// TIA Portal V15.1 export
// export: Created 2024-05-17T05:38:23.9003933Z, ExportSetting WithDefaults, DisplayName Totally Integrated Automation Portal, DisplayVersion V15.1 Update 5, DisplayName TIA Portal Openness, DisplayVersion V15.1 Update 5, DisplayName SINAMICS Startdrive Advanced, DisplayVersion V15.1, DisplayName G130, G150, S120, S150, SINAMICS MV, S210, DisplayVersion V15.1, DisplayName G110M, G120, G120C, G120D, G120P, DisplayVersion V15.1, DisplayName STEP 7 Professional, DisplayVersion V15.1 Update 5, DisplayName STEP 7 Safety, DisplayVersion V15.1, DisplayName WinCC Professional, DisplayVersion V15.1 Update 5, DisplayName SIMATIC Visualization Architect, DisplayVersion V15.1
FUNCTION "F209220ZS01Logic" : Void   // FC7021, F_FBD
TITLE = Safety Inputs ZMProc / Safety Logic 209220ZS01
{ S7_Optimized_Access := 'TRUE' }
VERSION : 0.1
// stored: AutoNumber false, IsIECCheckEnabled false, UDAEnableTagReadback false
   VAR_TEMP   // added for the SCL form of the ladder/FBD networks
      _w1 : Bool;
   END_VAR
BEGIN

REGION Network 1: **** 4.4 - Machine Status - Calculation **** Emergency Stop OK
   // Emergency Stop Ok When All Safety Inputs Are Ok
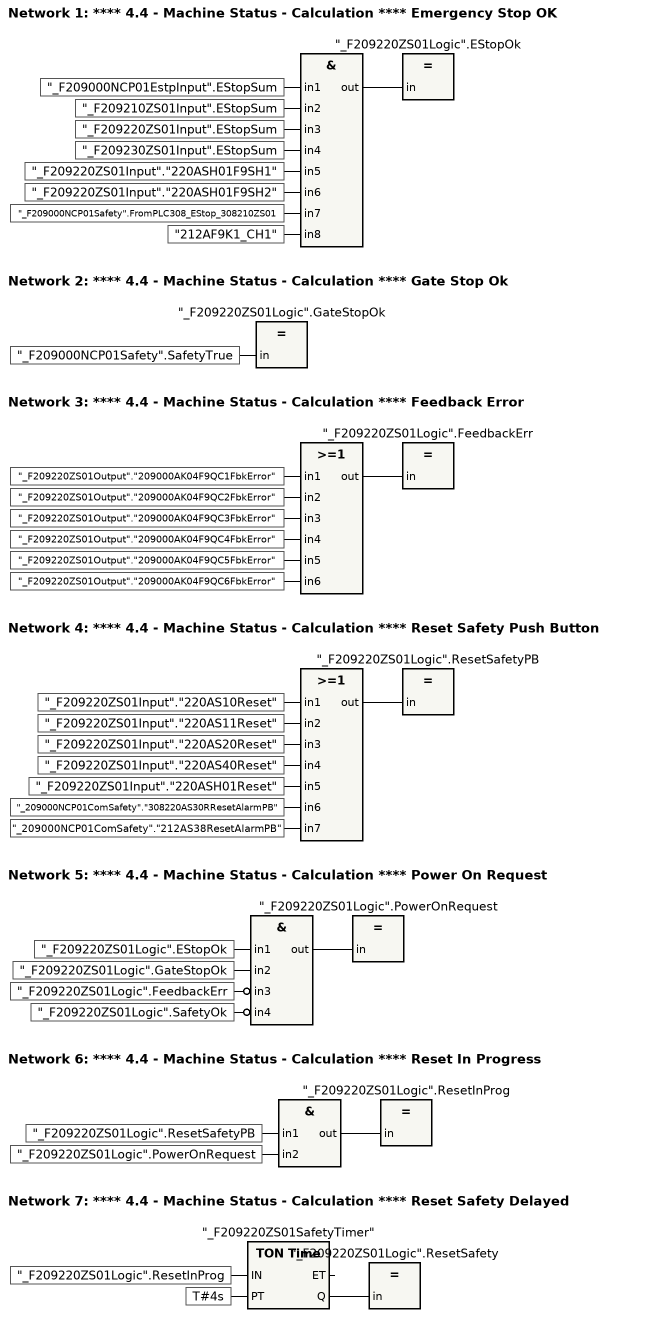
   "_F209220ZS01Logic".EStopOk := "_F209000NCP01EstpInput".EStopSum AND "_F209210ZS01Input".EStopSum AND "_F209220ZS01Input".EStopSum AND "_F209230ZS01Input".EStopSum AND "_F209220ZS01Input"."220ASH01F9SH1" AND "_F209220ZS01Input"."220ASH01F9SH2" AND "_F209000NCP01Safety".FromPLC308_EStop_308210ZS01 AND "212AF9K1_CH1";
END_REGION

REGION Network 2: **** 4.4 - Machine Status - Calculation **** Gate Stop Ok
   // Gate Stop Ok
   "_F209220ZS01Logic".GateStopOk := "_F209000NCP01Safety".SafetyTrue;
END_REGION

REGION Network 3: **** 4.4 - Machine Status - Calculation **** Feedback Error
   // Feedback Error
   "_F209220ZS01Logic".FeedbackErr := "_F209220ZS01Output"."209000AK04F9QC1FbkError" OR "_F209220ZS01Output"."209000AK04F9QC2FbkError" OR "_F209220ZS01Output"."209000AK04F9QC3FbkError" OR "_F209220ZS01Output"."209000AK04F9QC4FbkError" OR "_F209220ZS01Output"."209000AK04F9QC5FbkError" OR "_F209220ZS01Output"."209000AK04F9QC6FbkError";
END_REGION

REGION Network 4: **** 4.4 - Machine Status - Calculation **** Reset Safety Push Button
   // Reset Safety Push Button
   "_F209220ZS01Logic".ResetSafetyPB := "_F209220ZS01Input"."220AS10Reset" OR "_F209220ZS01Input"."220AS11Reset" OR "_F209220ZS01Input"."220AS20Reset" OR "_F209220ZS01Input"."220AS40Reset" OR "_F209220ZS01Input"."220ASH01Reset" OR "_209000NCP01ComSafety"."308220AS30RResetAlarmPB" OR "_209000NCP01ComSafety"."212AS38ResetAlarmPB";
END_REGION

REGION Network 5: **** 4.4 - Machine Status - Calculation **** Power On Request
   // Power On Request
   "_F209220ZS01Logic".PowerOnRequest := "_F209220ZS01Logic".EStopOk AND "_F209220ZS01Logic".GateStopOk AND NOT "_F209220ZS01Logic".FeedbackErr AND NOT "_F209220ZS01Logic".SafetyOk;
END_REGION

REGION Network 6: **** 4.4 - Machine Status - Calculation **** Reset In Progress
   // Reset In Progress
   "_F209220ZS01Logic".ResetInProg := "_F209220ZS01Logic".ResetSafetyPB AND "_F209220ZS01Logic".PowerOnRequest;
END_REGION

REGION Network 7: **** 4.4 - Machine Status - Calculation **** Reset Safety Delayed
   // Reset Safety Delayed
   "_F209220ZS01SafetyTimer".TON(IN := "_F209220ZS01Logic".ResetInProg, PT := T#4s);
   "_F209220ZS01Logic".ResetSafety := "_F209220ZS01SafetyTimer".Q;
END_REGION

REGION Network 8: **** 4.4 - Machine Status - Calculation **** Power On
   // Power On
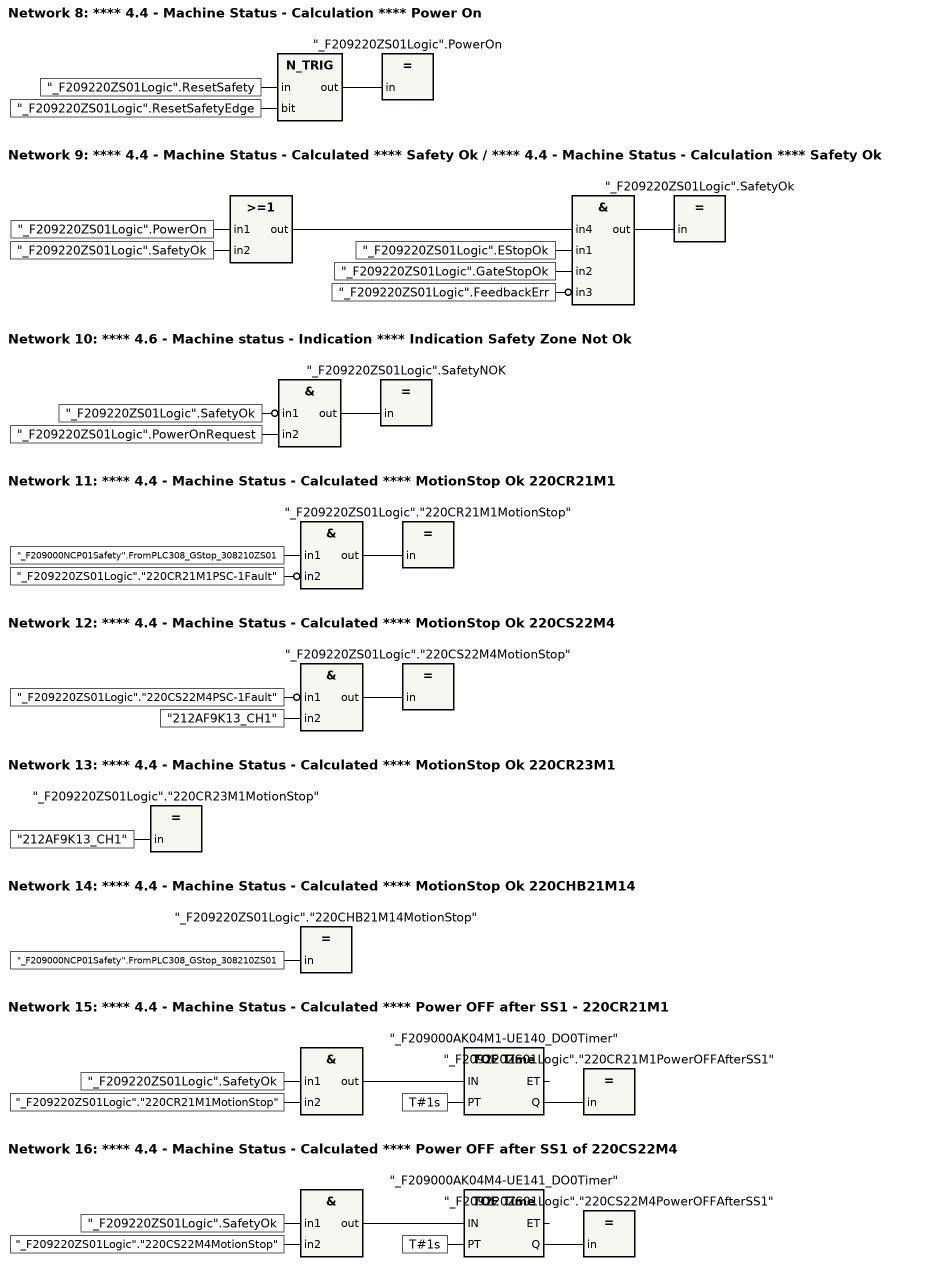
   #_w1 := NOT "_F209220ZS01Logic".ResetSafety AND "_F209220ZS01Logic".ResetSafetyEdge;   // falling edge
   "_F209220ZS01Logic".ResetSafetyEdge := "_F209220ZS01Logic".ResetSafety;
   "_F209220ZS01Logic".PowerOn := #_w1;
END_REGION

REGION Network 9: **** 4.4 - Machine Status - Calculated **** Safety Ok / **** 4.4 - Machine Status - Calculation **** Safety Ok
   // All safety is ok
   "_F209220ZS01Logic".SafetyOk := ("_F209220ZS01Logic".PowerOn OR "_F209220ZS01Logic".SafetyOk) AND "_F209220ZS01Logic".EStopOk AND "_F209220ZS01Logic".GateStopOk AND NOT "_F209220ZS01Logic".FeedbackErr;
END_REGION

REGION Network 10: **** 4.6 - Machine status - Indication **** Indication Safety Zone Not Ok
   // Indication Safety Zone Not Ok
   "_F209220ZS01Logic".SafetyNOK := NOT "_F209220ZS01Logic".SafetyOk AND "_F209220ZS01Logic".PowerOnRequest;
END_REGION

REGION Network 11: **** 4.4 - Machine Status - Calculated **** MotionStop Ok 220CR21M1
   // MotionStop Ok
   "_F209220ZS01Logic"."220CR21M1MotionStop" := "_F209000NCP01Safety".FromPLC308_GStop_308210ZS01 AND NOT "_F209220ZS01Logic"."220CR21M1PSC-1Fault";
END_REGION

REGION Network 12: **** 4.4 - Machine Status - Calculated **** MotionStop Ok 220CS22M4
   // MotionStop Ok
   "_F209220ZS01Logic"."220CS22M4MotionStop" := NOT "_F209220ZS01Logic"."220CS22M4PSC-1Fault" AND "212AF9K13_CH1";
END_REGION

REGION Network 13: **** 4.4 - Machine Status - Calculated **** MotionStop Ok 220CR23M1
   // MotionStop Ok
   "_F209220ZS01Logic"."220CR23M1MotionStop" := "212AF9K13_CH1";
END_REGION

REGION Network 14: **** 4.4 - Machine Status - Calculated **** MotionStop Ok 220CHB21M14
   // MotionStop Ok
   "_F209220ZS01Logic"."220CHB21M14MotionStop" := "_F209000NCP01Safety".FromPLC308_GStop_308210ZS01;
END_REGION

REGION Network 15: **** 4.4 - Machine Status - Calculated **** Power OFF after SS1 - 220CR21M1
   // SEW Drive Delay Power OFF
   "_F209000AK04M1-UE140_DO0Timer".TOF(IN := "_F209220ZS01Logic".SafetyOk AND "_F209220ZS01Logic"."220CR21M1MotionStop",
                           PT := T#1s);
   "_F209220ZS01Logic"."220CR21M1PowerOFFAfterSS1" := "_F209000AK04M1-UE140_DO0Timer".Q;
END_REGION

REGION Network 16: **** 4.4 - Machine Status - Calculated **** Power OFF after SS1 of 220CS22M4
   // SEW Drive Delay Power OFF
   "_F209000AK04M4-UE141_DO0Timer".TOF(IN := "_F209220ZS01Logic".SafetyOk AND "_F209220ZS01Logic"."220CS22M4MotionStop",
                           PT := T#1s);
   "_F209220ZS01Logic"."220CS22M4PowerOFFAfterSS1" := "_F209000AK04M4-UE141_DO0Timer".Q;
END_REGION

REGION Network 17: **** 4.4 - Machine Status - Calculated **** Power OFF after SS1 - 220CR23M1
   // SEW Drive Delay Power OFF
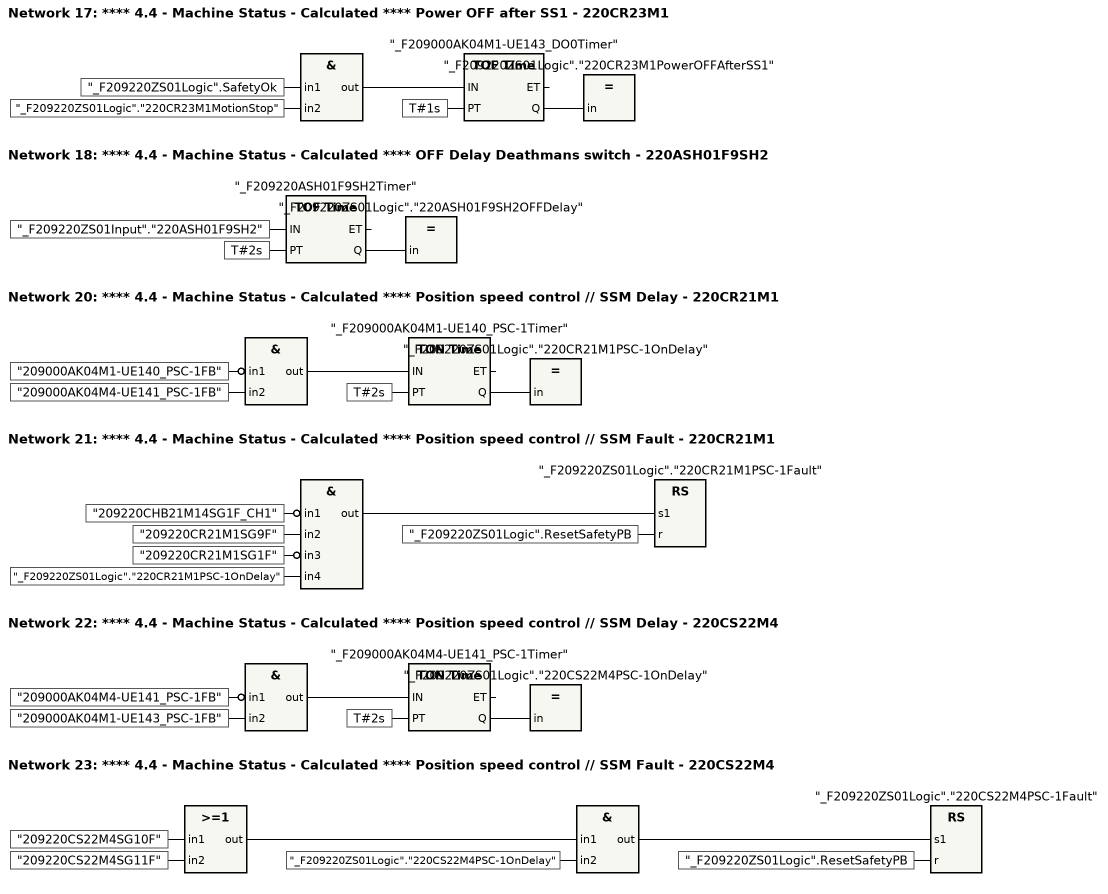
   "_F209000AK04M1-UE143_DO0Timer".TOF(IN := "_F209220ZS01Logic".SafetyOk AND "_F209220ZS01Logic"."220CR23M1MotionStop",
                           PT := T#1s);
   "_F209220ZS01Logic"."220CR23M1PowerOFFAfterSS1" := "_F209000AK04M1-UE143_DO0Timer".Q;
END_REGION

REGION Network 18: **** 4.4 - Machine Status - Calculated **** OFF Delay Deathmans switch - 220ASH01F9SH2
   "_F209220ASH01F9SH2Timer".TOF(IN := "_F209220ZS01Input"."220ASH01F9SH2", PT := T#2s);
   "_F209220ZS01Logic"."220ASH01F9SH2OFFDelay" := "_F209220ASH01F9SH2Timer".Q;
END_REGION

REGION Network 19: **** --------------------- SEW Safety Functions --------------------- ****
END_REGION

REGION Network 20: **** 4.4 - Machine Status - Calculated **** Position speed control // SSM Delay - 220CR21M1
   "_F209000AK04M1-UE140_PSC-1Timer".TON(IN := NOT "209000AK04M1-UE140_PSC-1FB" AND "209000AK04M4-UE141_PSC-1FB",
                           PT := T#2s);
   "_F209220ZS01Logic"."220CR21M1PSC-1OnDelay" := "_F209000AK04M1-UE140_PSC-1Timer".Q;
END_REGION

REGION Network 21: **** 4.4 - Machine Status - Calculated **** Position speed control // SSM Fault - 220CR21M1
   IF "_F209220ZS01Logic".ResetSafetyPB THEN
       "_F209220ZS01Logic"."220CR21M1PSC-1Fault" := FALSE;   // RS flip-flop
   END_IF;
   IF NOT "209220CHB21M14SG1F_CH1" AND "209220CR21M1SG9F" AND NOT "209220CR21M1SG1F" AND "_F209220ZS01Logic"."220CR21M1PSC-1OnDelay" THEN
       "_F209220ZS01Logic"."220CR21M1PSC-1Fault" := TRUE;
   END_IF;
END_REGION

REGION Network 22: **** 4.4 - Machine Status - Calculated **** Position speed control // SSM Delay - 220CS22M4
   "_F209000AK04M4-UE141_PSC-1Timer".TON(IN := NOT "209000AK04M4-UE141_PSC-1FB" AND "209000AK04M1-UE143_PSC-1FB",
                           PT := T#2s);
   "_F209220ZS01Logic"."220CS22M4PSC-1OnDelay" := "_F209000AK04M4-UE141_PSC-1Timer".Q;
END_REGION

REGION Network 23: **** 4.4 - Machine Status - Calculated **** Position speed control // SSM Fault - 220CS22M4
   IF "_F209220ZS01Logic".ResetSafetyPB THEN
       "_F209220ZS01Logic"."220CS22M4PSC-1Fault" := FALSE;   // RS flip-flop
   END_IF;
   IF ("209220CS22M4SG10F" OR "209220CS22M4SG11F") AND "_F209220ZS01Logic"."220CS22M4PSC-1OnDelay" THEN
       "_F209220ZS01Logic"."220CS22M4PSC-1Fault" := TRUE;
   END_IF;
END_REGION
END_FUNCTION
